// TIA Portal V16 export
// export: Created 2020-12-17T10:33:07.6875094Z, ExportSetting WithDefaults, WithReadOnly, DisplayName Totally Integrated Automation Portal, DisplayVersion V16 Update 2, DisplayName TIA Portal Version Control Interface, DisplayVersion V16 Update 2, DisplayName TIA Portal Openness, DisplayVersion V16 Update 2, DisplayName STEP 7 Professional, DisplayVersion V16 Update 2, DisplayName STEP 7 Safety, DisplayVersion V16, DisplayName WinCC Advanced / Unified PC, DisplayVersion V16 Update 2
DATA_BLOCK "XBlock_1_DB"   // DB2
{ S7_Optimized_Access := 'TRUE' }
VERSION : 0.1
// stored: AutoNumber true, CodeModifiedDate 2020-12-17T10:30:13.4748899Z, CompileDate 2020-12-17T10:32:57.5038962Z, CreationDate 2020-12-17T10:30:13.3967342Z, DBAccessibleFromOPCUA true, DownloadWithoutReinit false, InstanceOfName XBlock_1, InstanceOfNumber 1, InstanceOfType FB, InterfaceModifiedDate 2020-12-17T10:28:41.3528478Z, IsConsistent true, IsKnowHowProtected false, IsRetainMemResEnabled false, MemoryReserve 100, ModifiedDate 2020-12-17T10:30:13.4748899Z, ParameterModified 2020-12-17T10:28:41.3528478Z, StructureModified 2020-12-17T10:28:41.3528478Z, UDAEnableTagReadback false
"XBlock_1"
   // VAR_INPUT
   //    iEnable : Bool;
   //    iStart : Int;
   // END_VAR
   // VAR_OUTPUT
   //    qCounter : Int;
   // END_VAR
   // VAR
   //    sCounter : Int;
   // END_VAR
BEGIN
END_DATA_BLOCK
